Staubli VAL3: _toString.pgx

public program _toString(num x_nValue, string x_sFormat, string& x_string[])
  local num l_nPos
  local string l_string
begin
  l_string=toString(x_sFormat,x_nValue)
  l_nPos=find(l_string," ")
  if l_nPos!=-1
    x_string=delete(l_string,len(l_string)-l_nPos,l_nPos)
  else
    x_string=l_string
  endIf
end
